TYPE COMPLEX :
STRUCT
	re : REAL;
	im : REAL;
END_STRUCT
END_TYPE

(* stored: Version 1.1.0.1, ProductVersion 3.1.4022.7
   DUT COMPLEX: Id {9ba1b5bd-327a-4d98-a5e9-5112ec65a07c} *)
